TYPE ACREventCycleProp :
STRUCT
	_MemEventPos : DINT;
	_MemWriteCycle : UDINT;
END_STRUCT
END_TYPE

(* stored: Version 1.1.0.1, ProductVersion 3.1.4020.12
   DUT ACREventCycleProp: Id {6edec974-966b-424a-aa33-f1d9c1c71a1f} *)
